# EPICS substitutions: iocs/MC07/db/pmacStatus.substitutions
file "db/pmacStatus.db"
{
pattern
{SYS,             PMAC,    VERSION  PLC  PORT,  NAXES }
{"XF:06BMA-BI",   "MC:07", "1",     5,   "P0",  8     }
}
